// TIA Portal V15.1 export
// export: Created 2026-01-15T16:29:49.3065487Z, ExportSetting WithDefaults, WithReadOnly, DisplayName Totally Integrated Automation Portal, DisplayVersion V15.1 Update 8, DisplayName TIA Portal Openness, DisplayVersion V15.1 Update 8, DisplayName STEP 7 Professional, DisplayVersion V15.1 Update 8, DisplayName WinCC Advanced, DisplayVersion V15.1 Update 8
VAR_GLOBAL   // PLC tag table "Analog"
   AI_AG AT %IW68 : Int;
   AI_FD AT %IW70 : Int;
   AI_AP AT %IW72 : Int;
   AI_SB AT %IW74 : Int;
   AI_TEMP_TL AT %IW76 : Int;
   AI_TEMP_AG AT %IW78 : Int;
   AI_TEMP_TS AT %IW80 : Int;
   AI_TEMP_AP AT %IW82 : Int;
   BT_SPAN_Riasing AT %M2.0 : Bool;
   BT_ZERO_Raising AT %M2.1 : Bool;
   MANUAL_Raissing AT %M2.2 : Bool;
   AI_IND_AGG1 AT %IW100 : Int;
   AI_IND_AGG2 AT %IW102 : Int;
   AI_IND_AGG3 AT %IW104 : Int;
   AI_IND_AGG4 AT %IW106 : Int;
   AI_IND_AGG5 AT %IW108 : Int;
END_VAR
